ADAPTER IOthersValvesStatus (* Adapter Interface *)
  (* Standard: 61499-1 *)
  (* Version 0.0, 6/8/2026, Schneider Electric *)
  PACKAGE SE.Nereda;
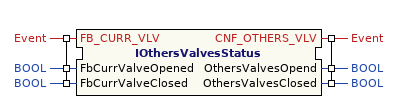
  EVENT_INPUT
    FB_CURR_VLV WITH FbCurrValveOpened, FbCurrValveClosed; (* Request from Socket *)
  END_EVENT
  EVENT_OUTPUT
    CNF_OTHERS_VLV WITH OthersValvesOpend, OthersValvesClosed; (* Confirmation from Plug *)
  END_EVENT
  VAR_INPUT
    FbCurrValveOpened : BOOL;
    FbCurrValveClosed : BOOL;
  END_VAR
  VAR_OUTPUT
    OthersValvesOpend : BOOL;
    OthersValvesClosed : BOOL;
  END_VAR
  SERVICE SOCKET/PLUG
    SEQUENCE request_confirm
      SOCKET.FB_CURR_VLV(REQD) -> PLUG.FB_CURR_VLV(REQD);
      PLUG.CNF_OTHERS_VLV(CNFD) -> SOCKET.CNF_OTHERS_VLV(CNFD);
    END_SEQUENCE
    SEQUENCE indication_response
      PLUG.IND(INDD) -> SOCKET.IND(INDD);
      SOCKET.RSP(RSPD) -> PLUG.RSP(RSPD);
    END_SEQUENCE
  END_SERVICE
END_ADAPTER
